{attribute addProperty BoxType "KL6224-0003"}
{attribute addProperty Id "StatusAT %I*UINT000Parameter_InAT %I*UDINT000State_Ch1AT %I*USINT000State_Ch2AT %I*USINT000State_Ch3AT %I*USINT000State_Ch4AT %I*USINT000Data_In_0AT %I*USINT000Data_In_1AT %I*USINT000Data_In_2AT %I*USINT000Data_In_3AT %I*USINT000Data_In_4AT %I*USINT000Data_In_5AT %I*USINT000Data_In_6AT %I*USINT000Data_In_7AT %I*USINT000Data_In_8AT %I*USINT000Data_In_9AT %I*USINT000Data_In_10AT %I*USINT000Data_In_11AT %I*USINT000Data_In_12AT %I*USINT000Data_In_13AT %I*USINT000Data_In_14AT %I*USINT000Data_In_15AT %I*USINT000Data_In_16AT %I*USINT000Data_In_17AT %I*USINT000Data_In_18AT %I*USINT000Data_In_19AT %I*USINT000Data_In_20AT %I*USINT000Data_In_21AT %I*USINT000Data_In_22AT %I*USINT000Data_In_23AT %I*USINT000Data_In_24AT %I*USINT000Data_In_25AT %I*USINT000Data_In_26AT %I*USINT000Data_In_27AT %I*USINT000Data_In_28AT %I*USINT000Data_In_29AT %I*USINT000Data_In_30AT %I*USINT000Data_In_31AT %I*USINT000Data_In_32AT %I*USINT000Data_In_33AT %I*USINT000Data_In_34AT %I*USINT000Data_In_35AT %I*USINT000Data_In_36AT %I*USINT000Data_In_37AT %I*USINT000ControlAT %Q*UINT000Parameter_OutAT %Q*UDINT000Data_Out_0AT %Q*USINT000Data_Out_1AT %Q*USINT000Data_Out_2AT %Q*USINT000Data_Out_3AT %Q*USINT000Data_Out_4AT %Q*USINT000Data_Out_5AT %Q*USINT000Data_Out_6AT %Q*USINT000Data_Out_7AT %Q*USINT000Data_Out_8AT %Q*USINT000Data_Out_9AT %Q*USINT000Data_Out_10AT %Q*USINT000Data_Out_11AT %Q*USINT000Data_Out_12AT %Q*USINT000Data_Out_13AT %Q*USINT000Data_Out_14AT %Q*USINT000Data_Out_15AT %Q*USINT000Data_Out_16AT %Q*USINT000Data_Out_17AT %Q*USINT000Data_Out_18AT %Q*USINT000Data_Out_19AT %Q*USINT000Data_Out_20AT %Q*USINT000Data_Out_21AT %Q*USINT000Data_Out_22AT %Q*USINT000Data_Out_23AT %Q*USINT000Data_Out_24AT %Q*USINT000Data_Out_25AT %Q*USINT000Data_Out_26AT %Q*USINT000Data_Out_27AT %Q*USINT000Data_Out_28AT %Q*USINT000Data_Out_29AT %Q*USINT000Data_Out_30AT %Q*USINT000Data_Out_31AT %Q*USINT000Data_Out_32AT %Q*USINT000Data_Out_33AT %Q*USINT000Data_Out_34AT %Q*USINT000Data_Out_35AT %Q*USINT000Data_Out_36AT %Q*USINT000Data_Out_37AT %Q*USINT000Data_Out_38AT %Q*USINT000Data_Out_39AT %Q*USINT000Data_Out_40AT %Q*USINT000Data_Out_41AT %Q*USINT000"}
{attribute addProperty CRC "68725328"}
{attribute addProperty SizeInBites "0"}
{attribute addProperty SizeInBytes "0"}
TYPE Channel_0418AA50 :
STRUCT
	{attribute addProperty Name "Status"}
	Status AT %I* : UINT;
	{attribute addProperty Name "Parameter_In"}
	Parameter_In AT %I* : UDINT;
	{attribute addProperty Name "State_Ch1"}
	State_Ch1 AT %I* : USINT;
	{attribute addProperty Name "State_Ch2"}
	State_Ch2 AT %I* : USINT;
	{attribute addProperty Name "State_Ch3"}
	State_Ch3 AT %I* : USINT;
	{attribute addProperty Name "State_Ch4"}
	State_Ch4 AT %I* : USINT;
	{attribute addProperty Name "Data_In_0"}
	Data_In_0 AT %I* : USINT;
	{attribute addProperty Name "Data_In_1"}
	Data_In_1 AT %I* : USINT;
	{attribute addProperty Name "Data_In_2"}
	Data_In_2 AT %I* : USINT;
	{attribute addProperty Name "Data_In_3"}
	Data_In_3 AT %I* : USINT;
	{attribute addProperty Name "Data_In_4"}
	Data_In_4 AT %I* : USINT;
	{attribute addProperty Name "Data_In_5"}
	Data_In_5 AT %I* : USINT;
	{attribute addProperty Name "Data_In_6"}
	Data_In_6 AT %I* : USINT;
	{attribute addProperty Name "Data_In_7"}
	Data_In_7 AT %I* : USINT;
	{attribute addProperty Name "Data_In_8"}
	Data_In_8 AT %I* : USINT;
	{attribute addProperty Name "Data_In_9"}
	Data_In_9 AT %I* : USINT;
	{attribute addProperty Name "Data_In_10"}
	Data_In_10 AT %I* : USINT;
	{attribute addProperty Name "Data_In_11"}
	Data_In_11 AT %I* : USINT;
	{attribute addProperty Name "Data_In_12"}
	Data_In_12 AT %I* : USINT;
	{attribute addProperty Name "Data_In_13"}
	Data_In_13 AT %I* : USINT;
	{attribute addProperty Name "Data_In_14"}
	Data_In_14 AT %I* : USINT;
	{attribute addProperty Name "Data_In_15"}
	Data_In_15 AT %I* : USINT;
	{attribute addProperty Name "Data_In_16"}
	Data_In_16 AT %I* : USINT;
	{attribute addProperty Name "Data_In_17"}
	Data_In_17 AT %I* : USINT;
	{attribute addProperty Name "Data_In_18"}
	Data_In_18 AT %I* : USINT;
	{attribute addProperty Name "Data_In_19"}
	Data_In_19 AT %I* : USINT;
	{attribute addProperty Name "Data_In_20"}
	Data_In_20 AT %I* : USINT;
	{attribute addProperty Name "Data_In_21"}
	Data_In_21 AT %I* : USINT;
	{attribute addProperty Name "Data_In_22"}
	Data_In_22 AT %I* : USINT;
	{attribute addProperty Name "Data_In_23"}
	Data_In_23 AT %I* : USINT;
	{attribute addProperty Name "Data_In_24"}
	Data_In_24 AT %I* : USINT;
	{attribute addProperty Name "Data_In_25"}
	Data_In_25 AT %I* : USINT;
	{attribute addProperty Name "Data_In_26"}
	Data_In_26 AT %I* : USINT;
	{attribute addProperty Name "Data_In_27"}
	Data_In_27 AT %I* : USINT;
	{attribute addProperty Name "Data_In_28"}
	Data_In_28 AT %I* : USINT;
	{attribute addProperty Name "Data_In_29"}
	Data_In_29 AT %I* : USINT;
	{attribute addProperty Name "Data_In_30"}
	Data_In_30 AT %I* : USINT;
	{attribute addProperty Name "Data_In_31"}
	Data_In_31 AT %I* : USINT;
	{attribute addProperty Name "Data_In_32"}
	Data_In_32 AT %I* : USINT;
	{attribute addProperty Name "Data_In_33"}
	Data_In_33 AT %I* : USINT;
	{attribute addProperty Name "Data_In_34"}
	Data_In_34 AT %I* : USINT;
	{attribute addProperty Name "Data_In_35"}
	Data_In_35 AT %I* : USINT;
	{attribute addProperty Name "Data_In_36"}
	Data_In_36 AT %I* : USINT;
	{attribute addProperty Name "Data_In_37"}
	Data_In_37 AT %I* : USINT;
	{attribute addProperty Name "Control"}
	Control AT %Q* : UINT;
	{attribute addProperty Name "Parameter_Out"}
	Parameter_Out AT %Q* : UDINT;
	{attribute addProperty Name "Data_Out_0"}
	Data_Out_0 AT %Q* : USINT;
	{attribute addProperty Name "Data_Out_1"}
	Data_Out_1 AT %Q* : USINT;
	{attribute addProperty Name "Data_Out_2"}
	Data_Out_2 AT %Q* : USINT;
	{attribute addProperty Name "Data_Out_3"}
	Data_Out_3 AT %Q* : USINT;
	{attribute addProperty Name "Data_Out_4"}
	Data_Out_4 AT %Q* : USINT;
	{attribute addProperty Name "Data_Out_5"}
	Data_Out_5 AT %Q* : USINT;
	{attribute addProperty Name "Data_Out_6"}
	Data_Out_6 AT %Q* : USINT;
	{attribute addProperty Name "Data_Out_7"}
	Data_Out_7 AT %Q* : USINT;
	{attribute addProperty Name "Data_Out_8"}
	Data_Out_8 AT %Q* : USINT;
	{attribute addProperty Name "Data_Out_9"}
	Data_Out_9 AT %Q* : USINT;
	{attribute addProperty Name "Data_Out_10"}
	Data_Out_10 AT %Q* : USINT;
	{attribute addProperty Name "Data_Out_11"}
	Data_Out_11 AT %Q* : USINT;
	{attribute addProperty Name "Data_Out_12"}
	Data_Out_12 AT %Q* : USINT;
	{attribute addProperty Name "Data_Out_13"}
	Data_Out_13 AT %Q* : USINT;
	{attribute addProperty Name "Data_Out_14"}
	Data_Out_14 AT %Q* : USINT;
	{attribute addProperty Name "Data_Out_15"}
	Data_Out_15 AT %Q* : USINT;
	{attribute addProperty Name "Data_Out_16"}
	Data_Out_16 AT %Q* : USINT;
	{attribute addProperty Name "Data_Out_17"}
	Data_Out_17 AT %Q* : USINT;
	{attribute addProperty Name "Data_Out_18"}
	Data_Out_18 AT %Q* : USINT;
	{attribute addProperty Name "Data_Out_19"}
	Data_Out_19 AT %Q* : USINT;
	{attribute addProperty Name "Data_Out_20"}
	Data_Out_20 AT %Q* : USINT;
	{attribute addProperty Name "Data_Out_21"}
	Data_Out_21 AT %Q* : USINT;
	{attribute addProperty Name "Data_Out_22"}
	Data_Out_22 AT %Q* : USINT;
	{attribute addProperty Name "Data_Out_23"}
	Data_Out_23 AT %Q* : USINT;
	{attribute addProperty Name "Data_Out_24"}
	Data_Out_24 AT %Q* : USINT;
	{attribute addProperty Name "Data_Out_25"}
	Data_Out_25 AT %Q* : USINT;
	{attribute addProperty Name "Data_Out_26"}
	Data_Out_26 AT %Q* : USINT;
	{attribute addProperty Name "Data_Out_27"}
	Data_Out_27 AT %Q* : USINT;
	{attribute addProperty Name "Data_Out_28"}
	Data_Out_28 AT %Q* : USINT;
	{attribute addProperty Name "Data_Out_29"}
	Data_Out_29 AT %Q* : USINT;
	{attribute addProperty Name "Data_Out_30"}
	Data_Out_30 AT %Q* : USINT;
	{attribute addProperty Name "Data_Out_31"}
	Data_Out_31 AT %Q* : USINT;
	{attribute addProperty Name "Data_Out_32"}
	Data_Out_32 AT %Q* : USINT;
	{attribute addProperty Name "Data_Out_33"}
	Data_Out_33 AT %Q* : USINT;
	{attribute addProperty Name "Data_Out_34"}
	Data_Out_34 AT %Q* : USINT;
	{attribute addProperty Name "Data_Out_35"}
	Data_Out_35 AT %Q* : USINT;
	{attribute addProperty Name "Data_Out_36"}
	Data_Out_36 AT %Q* : USINT;
	{attribute addProperty Name "Data_Out_37"}
	Data_Out_37 AT %Q* : USINT;
	{attribute addProperty Name "Data_Out_38"}
	Data_Out_38 AT %Q* : USINT;
	{attribute addProperty Name "Data_Out_39"}
	Data_Out_39 AT %Q* : USINT;
	{attribute addProperty Name "Data_Out_40"}
	Data_Out_40 AT %Q* : USINT;
	{attribute addProperty Name "Data_Out_41"}
	Data_Out_41 AT %Q* : USINT;
END_STRUCT
END_TYPE

(* stored: Version 1.2.0.0, ProductVersion 3.1.4024.9
   DUT Channel_0418AA50: Id {187cf373-ae30-4f63-87b9-4a8f49dc2fd6} *)
